// SIMATIC S7-200 project (STEP 7-Micro/WIN), CPU 224XP REL 02.01

SYMBOL_TABLE USER1
den_xe_vao       I0.2
den_xe_ra        I0.3
s_top            I0.1
barie            Q0.0
star             I0.0
reset            I0.4
den_bao_full     Q0.1
END_SYMBOL_TABLE

ORGANIZATION_BLOCK MAIN:OB1
TITLE=PROGRAM COMMENTS
BEGIN
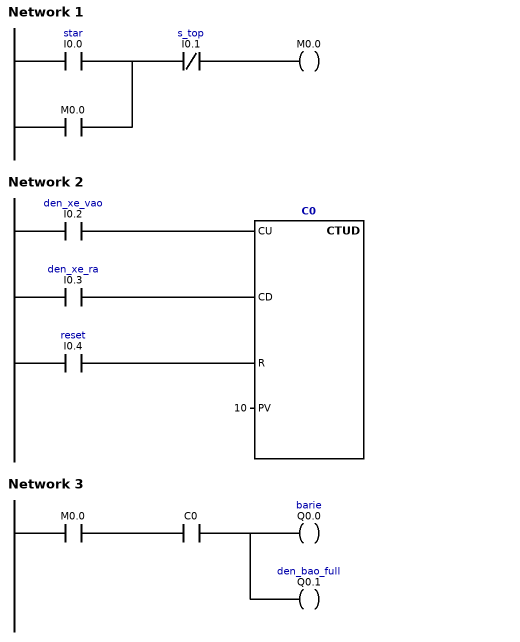
Network 1
LD     star:I0.0
O      M0.0
AN     s_top:I0.1
=      M0.0
Network 2
LD     den_xe_vao:I0.2
LD     den_xe_ra:I0.3
LD     reset:I0.4
CTUD   C0, 10
Network 3
LD     M0.0
A      C0
=      barie:Q0.0
=      den_bao_full:Q0.1
END_ORGANIZATION_BLOCK
